TYPE ST_AnyType :
STRUCT
	pValue : PVOID;
	nSize  : DINT;
	TypeClass : __SYSTEM.TYPE_CLASS;
END_STRUCT
END_TYPE

(* stored: Version 1.1.0.1
   DUT ST_AnyType: Id {5a7ba9f2-4a1b-41fd-97b7-9473bce2a8f4} *)
